FUNCTION_BLOCK DOWN_COUNT_TIMER
VAR_INPUT
	BOOL_SIGNAL_IN: BOOL;
	BOOL_TIMER_RST: BOOL;
	INT_AUTO_RST: INT;
	INT_SV_SEC: INT;
END_VAR
VAR_OUTPUT
	SIGNAL_BOOL: BOOL;
	PV_SEC_INT: INT;
END_VAR
VAR
	DF_1: R_TRIG;
	DF_2: R_TRIG;
	M1: BOOL;
	M2: BOOL;

	T100: TON;
	T101: TON;
	M100: BOOL;
	M101: BOOL;
	M200: BOOL;

	M110: BOOL;
	M300: BOOL;
END_VAR
VAR // added by the converter: edge detectors and wires of the graphical bodies
    _w1, _w2 : INT;
END_VAR

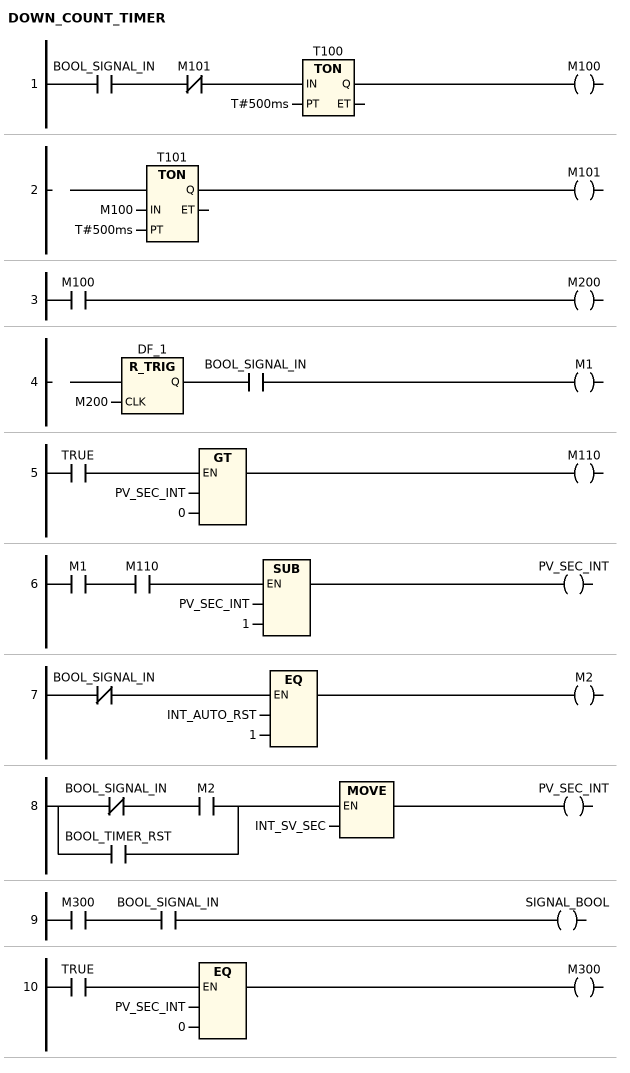
// NETWORK 1
T100(IN := BOOL_SIGNAL_IN AND NOT M101, PT := T#500ms); // TON
M100 := T100.Q;

// NETWORK 2
T101(IN := M100, PT := T#500ms); // TON
M101 := T101.Q;

// NETWORK 3
M200 := M100;

// NETWORK 4
DF_1(CLK := M200); // R_TRIG
M1 := DF_1.Q AND BOOL_SIGNAL_IN;

// NETWORK 5
M110 := PV_SEC_INT > 0;

// NETWORK 6
IF M1 AND M110 THEN _w1 := PV_SEC_INT - 1; END_IF
PV_SEC_INT := _w1;

// NETWORK 7
M2 := NOT BOOL_SIGNAL_IN AND INT_AUTO_RST = 1;

// NETWORK 8
IF NOT BOOL_SIGNAL_IN AND M2 OR BOOL_TIMER_RST THEN _w2 := INT_SV_SEC; END_IF
PV_SEC_INT := _w2;

// NETWORK 9
SIGNAL_BOOL := M300 AND BOOL_SIGNAL_IN;

// NETWORK 10
M300 := PV_SEC_INT = 0;

END_FUNCTION_BLOCK

(* stored: Version 1.1.0.1, ProductVersion 3.1.4024.12
   POU DOWN_COUNT_TIMER: Id {6901d3a2-378f-4470-8322-e307e3ab0a4f}, SpecialFunc None *)
